// TIA Portal V17 export
// export: Created 2023-03-24T09:45:04.5136241Z, ExportSetting None, DisplayName Totally Integrated Automation Portal, DisplayVersion V17 Update 4, DisplayName TIA Portal Openness, DisplayVersion V17 Update 4, DisplayName TIA Portal Version Control Interface, DisplayVersion V17, DisplayName STEP 7 Professional, DisplayVersion V17 Update 4, DisplayName STEP 7 Safety, DisplayVersion V17, DisplayName WinCC Advanced / Unified PC, DisplayVersion V17 Update 4
FUNCTION "FC_DI" : Void   // FC12, LAD
TITLE = FC_DI
{ S7_Optimized_Access := 'FALSE' }
// Digital Input
// stored: SetENOAutomatically false
BEGIN

REGION Network 1: DIGITAL INPUT 1
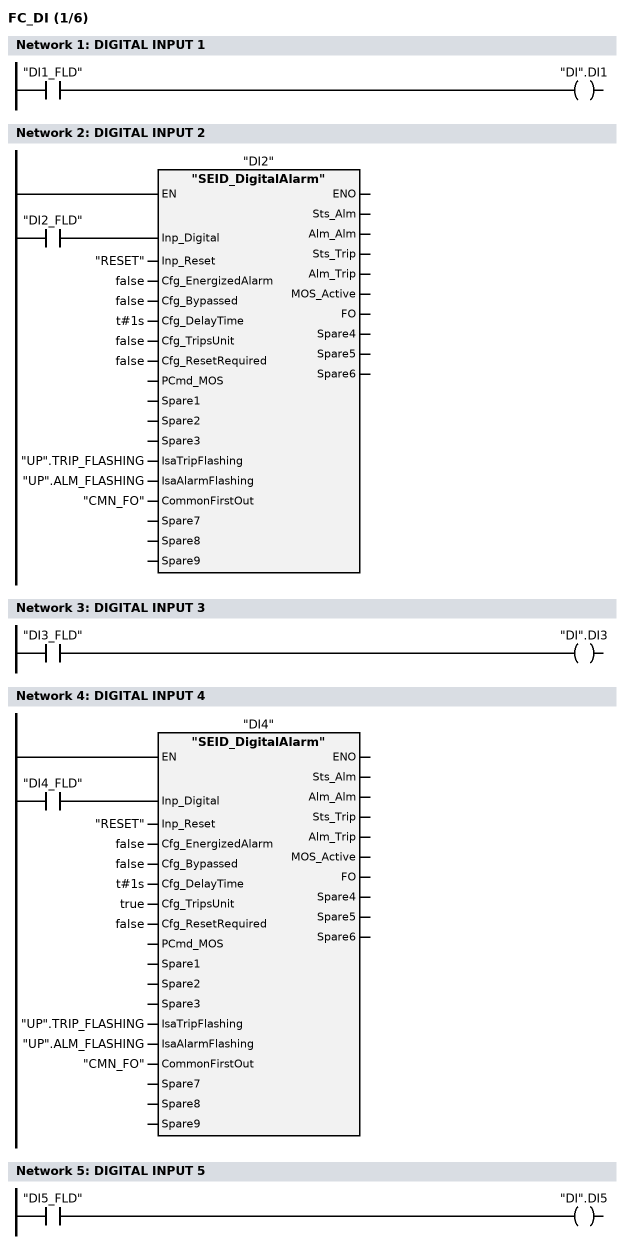
   RUNG wire#powerrail
      Contact( "DI1_FLD" )
      Coil( "DI".DI1 )
   END_RUNG
   // the same network as SCL:
   "DI".DI1 := "DI1_FLD";
END_REGION

REGION Network 2: DIGITAL INPUT 2
   RUNG wire#powerrail
      "DI2"(Inp_Digital := wire#w1, Inp_Reset := "RESET", Cfg_EnergizedAlarm := false, Cfg_Bypassed := false, Cfg_DelayTime := t#1s, Cfg_TripsUnit := false, Cfg_ResetRequired := false, PCmd_MOS :=, Spare1 :=, Spare2 :=, Spare3 :=, IsaTripFlashing := "UP".TRIP_FLASHING, IsaAlarmFlashing := "UP".ALM_FLASHING, CommonFirstOut := "CMN_FO", Spare7 :=, Spare8 :=, Spare9 :=, Sts_Alm =>, Alm_Alm =>, Sts_Trip =>, Alm_Trip =>, MOS_Active =>, FO =>, Spare4 =>, Spare5 =>, Spare6 =>)
   END_RUNG
   RUNG wire#powerrail
      Contact( "DI2_FLD" )
   END_RUNG wire#w1
   // the same network as SCL:
   "DI2"(Inp_Digital := "DI2_FLD",   // "SEID_DigitalAlarm"
         Inp_Reset := "RESET",
         Cfg_EnergizedAlarm := false,
         Cfg_Bypassed := false,
         Cfg_DelayTime := t#1s,
         Cfg_TripsUnit := false,
         Cfg_ResetRequired := false,
         IsaTripFlashing := "UP".TRIP_FLASHING,
         IsaAlarmFlashing := "UP".ALM_FLASHING,
         CommonFirstOut := "CMN_FO");
END_REGION

REGION Network 3: DIGITAL INPUT 3
   RUNG wire#powerrail
      Contact( "DI3_FLD" )
      Coil( "DI".DI3 )
   END_RUNG
   // the same network as SCL:
   "DI".DI3 := "DI3_FLD";
END_REGION

REGION Network 4: DIGITAL INPUT 4
   RUNG wire#powerrail
      "DI4"(Inp_Digital := wire#w1, Inp_Reset := "RESET", Cfg_EnergizedAlarm := false, Cfg_Bypassed := false, Cfg_DelayTime := t#1s, Cfg_TripsUnit := true, Cfg_ResetRequired := false, PCmd_MOS :=, Spare1 :=, Spare2 :=, Spare3 :=, IsaTripFlashing := "UP".TRIP_FLASHING, IsaAlarmFlashing := "UP".ALM_FLASHING, CommonFirstOut := "CMN_FO", Spare7 :=, Spare8 :=, Spare9 :=, Sts_Alm =>, Alm_Alm =>, Sts_Trip =>, Alm_Trip =>, MOS_Active =>, FO =>, Spare4 =>, Spare5 =>, Spare6 =>)
   END_RUNG
   RUNG wire#powerrail
      Contact( "DI4_FLD" )
   END_RUNG wire#w1
   // the same network as SCL:
   "DI4"(Inp_Digital := "DI4_FLD",   // "SEID_DigitalAlarm"
         Inp_Reset := "RESET",
         Cfg_EnergizedAlarm := false,
         Cfg_Bypassed := false,
         Cfg_DelayTime := t#1s,
         Cfg_TripsUnit := true,
         Cfg_ResetRequired := false,
         IsaTripFlashing := "UP".TRIP_FLASHING,
         IsaAlarmFlashing := "UP".ALM_FLASHING,
         CommonFirstOut := "CMN_FO");
END_REGION

REGION Network 5: DIGITAL INPUT 5
   RUNG wire#powerrail
      Contact( "DI5_FLD" )
      Coil( "DI".DI5 )
   END_RUNG
   // the same network as SCL:
   "DI".DI5 := "DI5_FLD";
END_REGION

REGION Network 6: DIGITAL INPUT 6
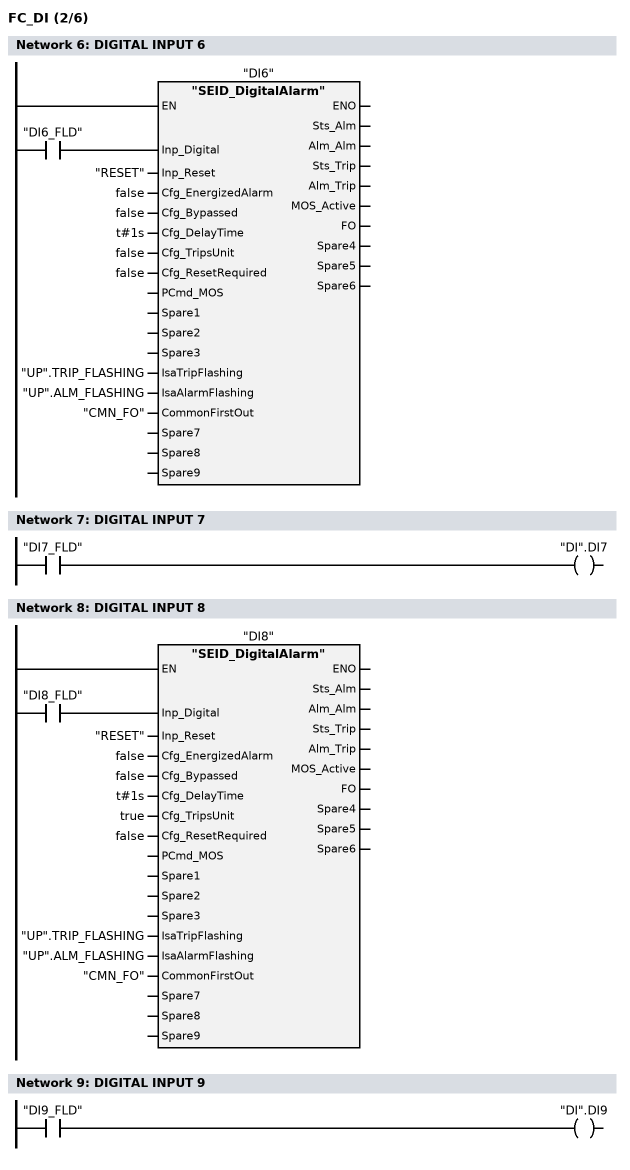
   RUNG wire#powerrail
      "DI6"(Inp_Digital := wire#w1, Inp_Reset := "RESET", Cfg_EnergizedAlarm := false, Cfg_Bypassed := false, Cfg_DelayTime := t#1s, Cfg_TripsUnit := false, Cfg_ResetRequired := false, PCmd_MOS :=, Spare1 :=, Spare2 :=, Spare3 :=, IsaTripFlashing := "UP".TRIP_FLASHING, IsaAlarmFlashing := "UP".ALM_FLASHING, CommonFirstOut := "CMN_FO", Spare7 :=, Spare8 :=, Spare9 :=, Sts_Alm =>, Alm_Alm =>, Sts_Trip =>, Alm_Trip =>, MOS_Active =>, FO =>, Spare4 =>, Spare5 =>, Spare6 =>)
   END_RUNG
   RUNG wire#powerrail
      Contact( "DI6_FLD" )
   END_RUNG wire#w1
   // the same network as SCL:
   "DI6"(Inp_Digital := "DI6_FLD",   // "SEID_DigitalAlarm"
         Inp_Reset := "RESET",
         Cfg_EnergizedAlarm := false,
         Cfg_Bypassed := false,
         Cfg_DelayTime := t#1s,
         Cfg_TripsUnit := false,
         Cfg_ResetRequired := false,
         IsaTripFlashing := "UP".TRIP_FLASHING,
         IsaAlarmFlashing := "UP".ALM_FLASHING,
         CommonFirstOut := "CMN_FO");
END_REGION

REGION Network 7: DIGITAL INPUT 7
   RUNG wire#powerrail
      Contact( "DI7_FLD" )
      Coil( "DI".DI7 )
   END_RUNG
   // the same network as SCL:
   "DI".DI7 := "DI7_FLD";
END_REGION

REGION Network 8: DIGITAL INPUT 8
   RUNG wire#powerrail
      "DI8"(Inp_Digital := wire#w1, Inp_Reset := "RESET", Cfg_EnergizedAlarm := false, Cfg_Bypassed := false, Cfg_DelayTime := t#1s, Cfg_TripsUnit := true, Cfg_ResetRequired := false, PCmd_MOS :=, Spare1 :=, Spare2 :=, Spare3 :=, IsaTripFlashing := "UP".TRIP_FLASHING, IsaAlarmFlashing := "UP".ALM_FLASHING, CommonFirstOut := "CMN_FO", Spare7 :=, Spare8 :=, Spare9 :=, Sts_Alm =>, Alm_Alm =>, Sts_Trip =>, Alm_Trip =>, MOS_Active =>, FO =>, Spare4 =>, Spare5 =>, Spare6 =>)
   END_RUNG
   RUNG wire#powerrail
      Contact( "DI8_FLD" )
   END_RUNG wire#w1
   // the same network as SCL:
   "DI8"(Inp_Digital := "DI8_FLD",   // "SEID_DigitalAlarm"
         Inp_Reset := "RESET",
         Cfg_EnergizedAlarm := false,
         Cfg_Bypassed := false,
         Cfg_DelayTime := t#1s,
         Cfg_TripsUnit := true,
         Cfg_ResetRequired := false,
         IsaTripFlashing := "UP".TRIP_FLASHING,
         IsaAlarmFlashing := "UP".ALM_FLASHING,
         CommonFirstOut := "CMN_FO");
END_REGION

REGION Network 9: DIGITAL INPUT 9
   RUNG wire#powerrail
      Contact( "DI9_FLD" )
      Coil( "DI".DI9 )
   END_RUNG
   // the same network as SCL:
   "DI".DI9 := "DI9_FLD";
END_REGION

REGION Network 10: DIGITAL INPUT 10
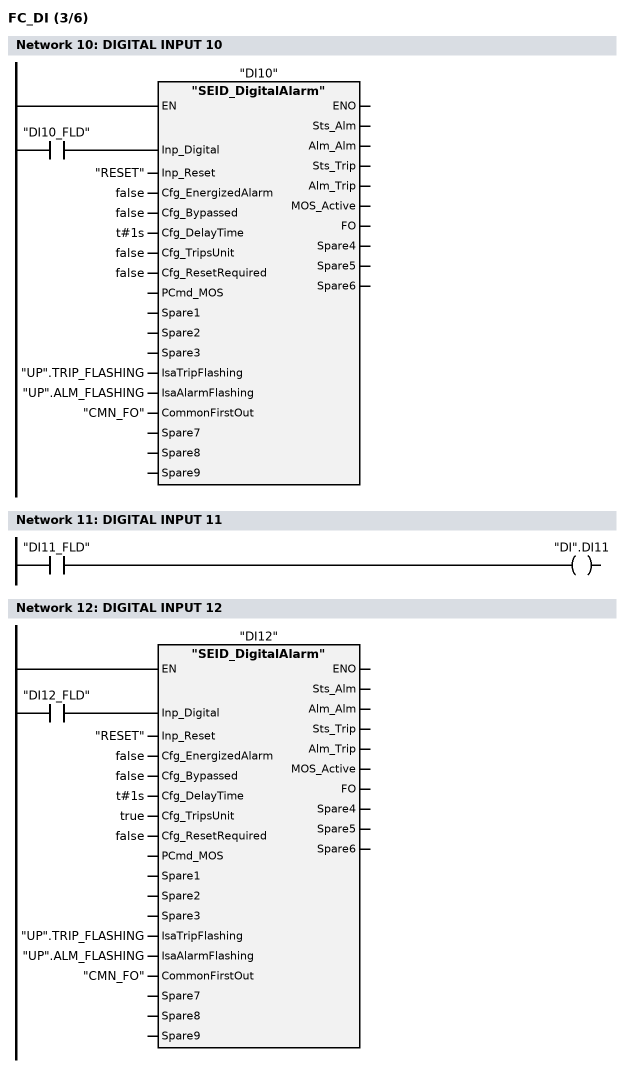
   RUNG wire#powerrail
      "DI10"(Inp_Digital := wire#w1, Inp_Reset := "RESET", Cfg_EnergizedAlarm := false, Cfg_Bypassed := false, Cfg_DelayTime := t#1s, Cfg_TripsUnit := false, Cfg_ResetRequired := false, PCmd_MOS :=, Spare1 :=, Spare2 :=, Spare3 :=, IsaTripFlashing := "UP".TRIP_FLASHING, IsaAlarmFlashing := "UP".ALM_FLASHING, CommonFirstOut := "CMN_FO", Spare7 :=, Spare8 :=, Spare9 :=, Sts_Alm =>, Alm_Alm =>, Sts_Trip =>, Alm_Trip =>, MOS_Active =>, FO =>, Spare4 =>, Spare5 =>, Spare6 =>)
   END_RUNG
   RUNG wire#powerrail
      Contact( "DI10_FLD" )
   END_RUNG wire#w1
   // the same network as SCL:
   "DI10"(Inp_Digital := "DI10_FLD",   // "SEID_DigitalAlarm"
          Inp_Reset := "RESET",
          Cfg_EnergizedAlarm := false,
          Cfg_Bypassed := false,
          Cfg_DelayTime := t#1s,
          Cfg_TripsUnit := false,
          Cfg_ResetRequired := false,
          IsaTripFlashing := "UP".TRIP_FLASHING,
          IsaAlarmFlashing := "UP".ALM_FLASHING,
          CommonFirstOut := "CMN_FO");
END_REGION

REGION Network 11: DIGITAL INPUT 11
   RUNG wire#powerrail
      Contact( "DI11_FLD" )
      Coil( "DI".DI11 )
   END_RUNG
   // the same network as SCL:
   "DI".DI11 := "DI11_FLD";
END_REGION

REGION Network 12: DIGITAL INPUT 12
   RUNG wire#powerrail
      "DI12"(Inp_Digital := wire#w1, Inp_Reset := "RESET", Cfg_EnergizedAlarm := false, Cfg_Bypassed := false, Cfg_DelayTime := t#1s, Cfg_TripsUnit := true, Cfg_ResetRequired := false, PCmd_MOS :=, Spare1 :=, Spare2 :=, Spare3 :=, IsaTripFlashing := "UP".TRIP_FLASHING, IsaAlarmFlashing := "UP".ALM_FLASHING, CommonFirstOut := "CMN_FO", Spare7 :=, Spare8 :=, Spare9 :=, Sts_Alm =>, Alm_Alm =>, Sts_Trip =>, Alm_Trip =>, MOS_Active =>, FO =>, Spare4 =>, Spare5 =>, Spare6 =>)
   END_RUNG
   RUNG wire#powerrail
      Contact( "DI12_FLD" )
   END_RUNG wire#w1
   // the same network as SCL:
   "DI12"(Inp_Digital := "DI12_FLD",   // "SEID_DigitalAlarm"
          Inp_Reset := "RESET",
          Cfg_EnergizedAlarm := false,
          Cfg_Bypassed := false,
          Cfg_DelayTime := t#1s,
          Cfg_TripsUnit := true,
          Cfg_ResetRequired := false,
          IsaTripFlashing := "UP".TRIP_FLASHING,
          IsaAlarmFlashing := "UP".ALM_FLASHING,
          CommonFirstOut := "CMN_FO");
END_REGION

REGION Network 13: DIGITAL INPUT 13
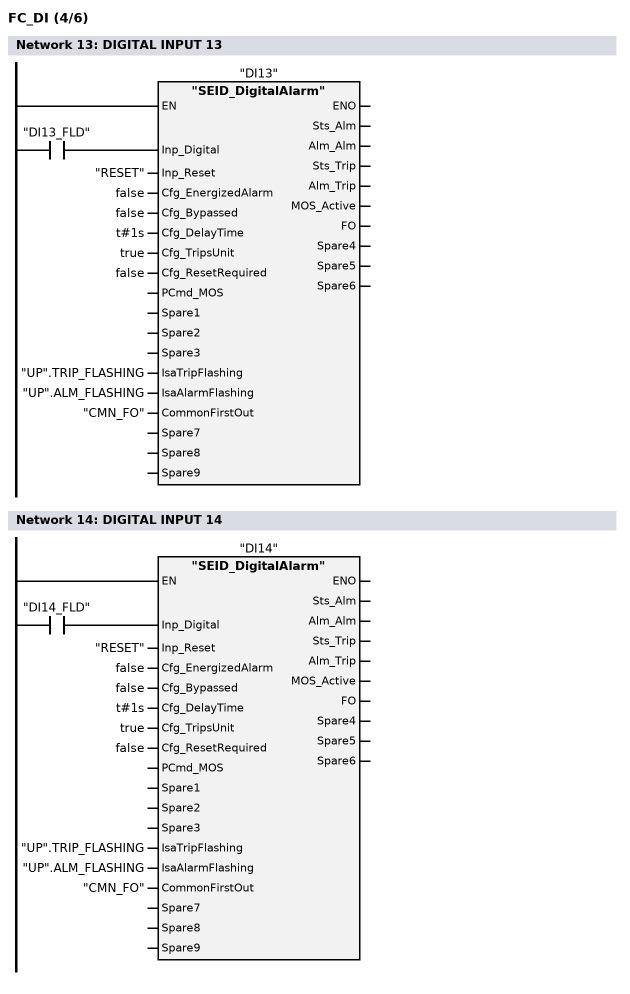
   RUNG wire#powerrail
      "DI13"(Inp_Digital := wire#w1, Inp_Reset := "RESET", Cfg_EnergizedAlarm := false, Cfg_Bypassed := false, Cfg_DelayTime := t#1s, Cfg_TripsUnit := true, Cfg_ResetRequired := false, PCmd_MOS :=, Spare1 :=, Spare2 :=, Spare3 :=, IsaTripFlashing := "UP".TRIP_FLASHING, IsaAlarmFlashing := "UP".ALM_FLASHING, CommonFirstOut := "CMN_FO", Spare7 :=, Spare8 :=, Spare9 :=, Sts_Alm =>, Alm_Alm =>, Sts_Trip =>, Alm_Trip =>, MOS_Active =>, FO =>, Spare4 =>, Spare5 =>, Spare6 =>)
   END_RUNG
   RUNG wire#powerrail
      Contact( "DI13_FLD" )
   END_RUNG wire#w1
   // the same network as SCL:
   "DI13"(Inp_Digital := "DI13_FLD",   // "SEID_DigitalAlarm"
          Inp_Reset := "RESET",
          Cfg_EnergizedAlarm := false,
          Cfg_Bypassed := false,
          Cfg_DelayTime := t#1s,
          Cfg_TripsUnit := true,
          Cfg_ResetRequired := false,
          IsaTripFlashing := "UP".TRIP_FLASHING,
          IsaAlarmFlashing := "UP".ALM_FLASHING,
          CommonFirstOut := "CMN_FO");
END_REGION

REGION Network 14: DIGITAL INPUT 14
   RUNG wire#powerrail
      "DI14"(Inp_Digital := wire#w1, Inp_Reset := "RESET", Cfg_EnergizedAlarm := false, Cfg_Bypassed := false, Cfg_DelayTime := t#1s, Cfg_TripsUnit := true, Cfg_ResetRequired := false, PCmd_MOS :=, Spare1 :=, Spare2 :=, Spare3 :=, IsaTripFlashing := "UP".TRIP_FLASHING, IsaAlarmFlashing := "UP".ALM_FLASHING, CommonFirstOut := "CMN_FO", Spare7 :=, Spare8 :=, Spare9 :=, Sts_Alm =>, Alm_Alm =>, Sts_Trip =>, Alm_Trip =>, MOS_Active =>, FO =>, Spare4 =>, Spare5 =>, Spare6 =>)
   END_RUNG
   RUNG wire#powerrail
      Contact( "DI14_FLD" )
   END_RUNG wire#w1
   // the same network as SCL:
   "DI14"(Inp_Digital := "DI14_FLD",   // "SEID_DigitalAlarm"
          Inp_Reset := "RESET",
          Cfg_EnergizedAlarm := false,
          Cfg_Bypassed := false,
          Cfg_DelayTime := t#1s,
          Cfg_TripsUnit := true,
          Cfg_ResetRequired := false,
          IsaTripFlashing := "UP".TRIP_FLASHING,
          IsaAlarmFlashing := "UP".ALM_FLASHING,
          CommonFirstOut := "CMN_FO");
END_REGION

REGION Network 15: DIGITAL INPUT 15
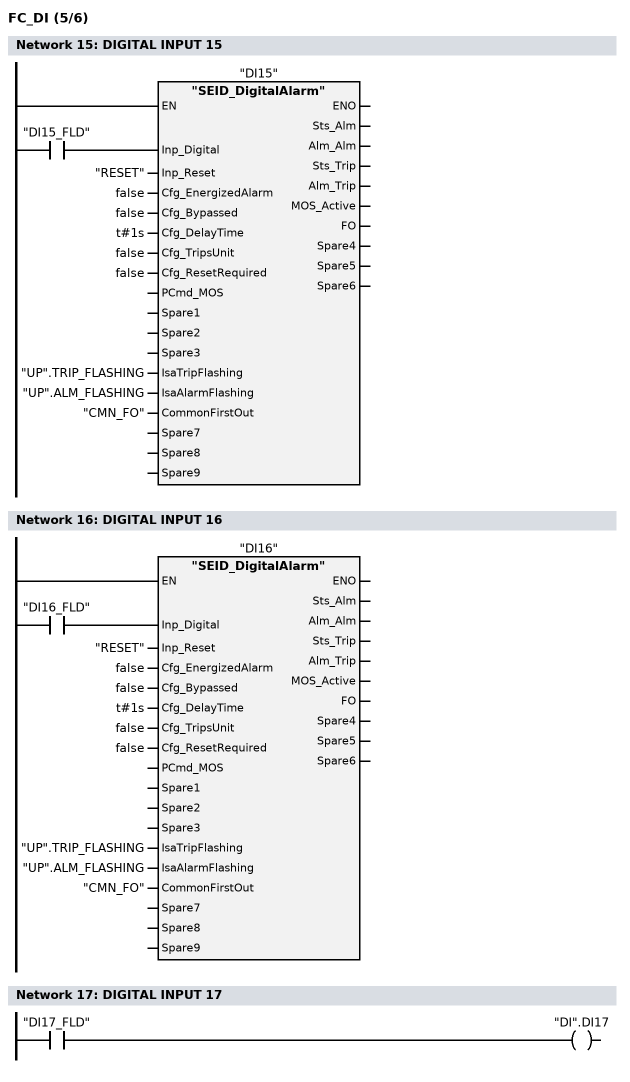
   RUNG wire#powerrail
      "DI15"(Inp_Digital := wire#w1, Inp_Reset := "RESET", Cfg_EnergizedAlarm := false, Cfg_Bypassed := false, Cfg_DelayTime := t#1s, Cfg_TripsUnit := false, Cfg_ResetRequired := false, PCmd_MOS :=, Spare1 :=, Spare2 :=, Spare3 :=, IsaTripFlashing := "UP".TRIP_FLASHING, IsaAlarmFlashing := "UP".ALM_FLASHING, CommonFirstOut := "CMN_FO", Spare7 :=, Spare8 :=, Spare9 :=, Sts_Alm =>, Alm_Alm =>, Sts_Trip =>, Alm_Trip =>, MOS_Active =>, FO =>, Spare4 =>, Spare5 =>, Spare6 =>)
   END_RUNG
   RUNG wire#powerrail
      Contact( "DI15_FLD" )
   END_RUNG wire#w1
   // the same network as SCL:
   "DI15"(Inp_Digital := "DI15_FLD",   // "SEID_DigitalAlarm"
          Inp_Reset := "RESET",
          Cfg_EnergizedAlarm := false,
          Cfg_Bypassed := false,
          Cfg_DelayTime := t#1s,
          Cfg_TripsUnit := false,
          Cfg_ResetRequired := false,
          IsaTripFlashing := "UP".TRIP_FLASHING,
          IsaAlarmFlashing := "UP".ALM_FLASHING,
          CommonFirstOut := "CMN_FO");
END_REGION

REGION Network 16: DIGITAL INPUT 16
   RUNG wire#powerrail
      "DI16"(Inp_Digital := wire#w1, Inp_Reset := "RESET", Cfg_EnergizedAlarm := false, Cfg_Bypassed := false, Cfg_DelayTime := t#1s, Cfg_TripsUnit := false, Cfg_ResetRequired := false, PCmd_MOS :=, Spare1 :=, Spare2 :=, Spare3 :=, IsaTripFlashing := "UP".TRIP_FLASHING, IsaAlarmFlashing := "UP".ALM_FLASHING, CommonFirstOut := "CMN_FO", Spare7 :=, Spare8 :=, Spare9 :=, Sts_Alm =>, Alm_Alm =>, Sts_Trip =>, Alm_Trip =>, MOS_Active =>, FO =>, Spare4 =>, Spare5 =>, Spare6 =>)
   END_RUNG
   RUNG wire#powerrail
      Contact( "DI16_FLD" )
   END_RUNG wire#w1
   // the same network as SCL:
   "DI16"(Inp_Digital := "DI16_FLD",   // "SEID_DigitalAlarm"
          Inp_Reset := "RESET",
          Cfg_EnergizedAlarm := false,
          Cfg_Bypassed := false,
          Cfg_DelayTime := t#1s,
          Cfg_TripsUnit := false,
          Cfg_ResetRequired := false,
          IsaTripFlashing := "UP".TRIP_FLASHING,
          IsaAlarmFlashing := "UP".ALM_FLASHING,
          CommonFirstOut := "CMN_FO");
END_REGION

REGION Network 17: DIGITAL INPUT 17
   RUNG wire#powerrail
      Contact( "DI17_FLD" )
      Coil( "DI".DI17 )
   END_RUNG
   // the same network as SCL:
   "DI".DI17 := "DI17_FLD";
END_REGION

REGION Network 18: DIGITAL INPUT 18
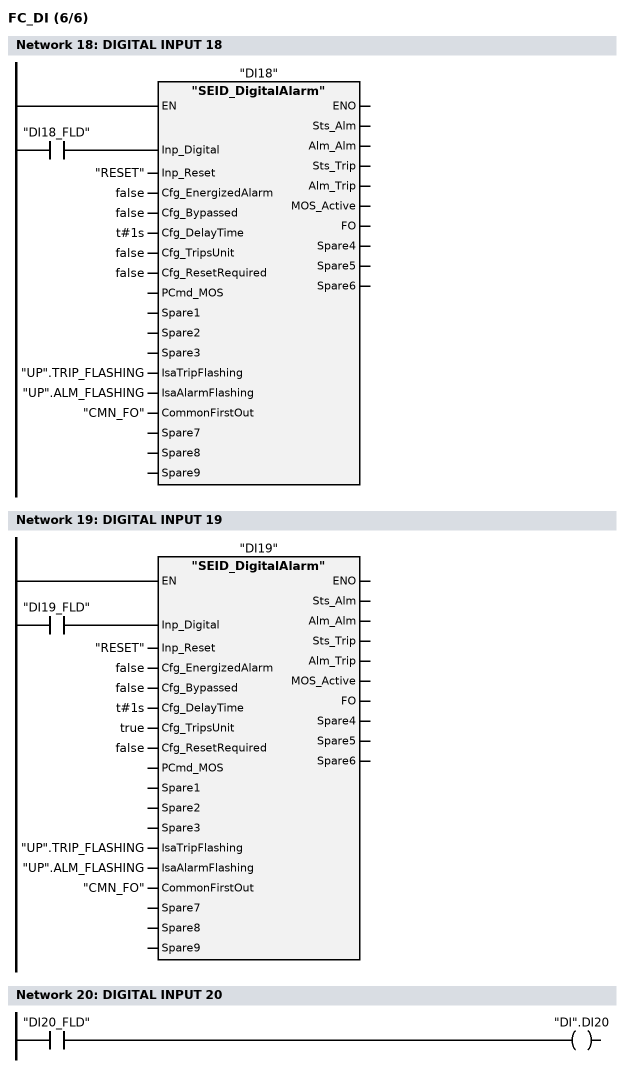
   RUNG wire#powerrail
      "DI18"(Inp_Digital := wire#w1, Inp_Reset := "RESET", Cfg_EnergizedAlarm := false, Cfg_Bypassed := false, Cfg_DelayTime := t#1s, Cfg_TripsUnit := false, Cfg_ResetRequired := false, PCmd_MOS :=, Spare1 :=, Spare2 :=, Spare3 :=, IsaTripFlashing := "UP".TRIP_FLASHING, IsaAlarmFlashing := "UP".ALM_FLASHING, CommonFirstOut := "CMN_FO", Spare7 :=, Spare8 :=, Spare9 :=, Sts_Alm =>, Alm_Alm =>, Sts_Trip =>, Alm_Trip =>, MOS_Active =>, FO =>, Spare4 =>, Spare5 =>, Spare6 =>)
   END_RUNG
   RUNG wire#powerrail
      Contact( "DI18_FLD" )
   END_RUNG wire#w1
   // the same network as SCL:
   "DI18"(Inp_Digital := "DI18_FLD",   // "SEID_DigitalAlarm"
          Inp_Reset := "RESET",
          Cfg_EnergizedAlarm := false,
          Cfg_Bypassed := false,
          Cfg_DelayTime := t#1s,
          Cfg_TripsUnit := false,
          Cfg_ResetRequired := false,
          IsaTripFlashing := "UP".TRIP_FLASHING,
          IsaAlarmFlashing := "UP".ALM_FLASHING,
          CommonFirstOut := "CMN_FO");
END_REGION

REGION Network 19: DIGITAL INPUT 19
   RUNG wire#powerrail
      "DI19"(Inp_Digital := wire#w1, Inp_Reset := "RESET", Cfg_EnergizedAlarm := false, Cfg_Bypassed := false, Cfg_DelayTime := t#1s, Cfg_TripsUnit := true, Cfg_ResetRequired := false, PCmd_MOS :=, Spare1 :=, Spare2 :=, Spare3 :=, IsaTripFlashing := "UP".TRIP_FLASHING, IsaAlarmFlashing := "UP".ALM_FLASHING, CommonFirstOut := "CMN_FO", Spare7 :=, Spare8 :=, Spare9 :=, Sts_Alm =>, Alm_Alm =>, Sts_Trip =>, Alm_Trip =>, MOS_Active =>, FO =>, Spare4 =>, Spare5 =>, Spare6 =>)
   END_RUNG
   RUNG wire#powerrail
      Contact( "DI19_FLD" )
   END_RUNG wire#w1
   // the same network as SCL:
   "DI19"(Inp_Digital := "DI19_FLD",   // "SEID_DigitalAlarm"
          Inp_Reset := "RESET",
          Cfg_EnergizedAlarm := false,
          Cfg_Bypassed := false,
          Cfg_DelayTime := t#1s,
          Cfg_TripsUnit := true,
          Cfg_ResetRequired := false,
          IsaTripFlashing := "UP".TRIP_FLASHING,
          IsaAlarmFlashing := "UP".ALM_FLASHING,
          CommonFirstOut := "CMN_FO");
END_REGION

REGION Network 20: DIGITAL INPUT 20
   RUNG wire#powerrail
      Contact( "DI20_FLD" )
      Coil( "DI".DI20 )
   END_RUNG
   // the same network as SCL:
   "DI".DI20 := "DI20_FLD";
END_REGION
END_FUNCTION
